FUNCTION_BLOCK LT_TIME (* IEC 61131-3,Table 28#9 *)
  (* Standard: 61131-3 *)
  (* Version 0.0, 2004-12-15, JHC, Rockwell Automation, Converted from SRC format. *)
  (* Compiler header: package fb.rt.plc.comp; *)
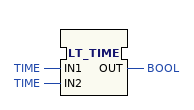
  VAR_INPUT
    IN1 : TIME;
    IN2 : TIME;
  END_VAR
  VAR_OUTPUT
    OUT : BOOL;
  END_VAR
END_FUNCTION_BLOCK
